// TIA Portal project "XSFW_TIA15.133301_A0" (V15.1)

(* hardware
DEVICE "S7-1200 station_1"  S7-1200 Station
   slot 0: "Rack_0"  S7-1200 Rack  Rack  V1.0
   slot 1: "PLC_1"  CPU 1214C DC/DC/DC  6ES7 214-1AG40-0XB0  V4.3
   slot 2: "DI 16x24VDC_1"  6ES7 221-1BH32-0XB0  V2.0
   slot 3: "DI 16x24VDC_2"  6ES7 221-1BH32-0XB0  V2.0
   slot 4: "DQ 16x24VDC_1"  SM 1222 DQ16 x 24VDC  6ES7 222-1BH32-0XB0  V2.0
*)

// ===== PLC "PLC_1"  CPU 1214C DC/DC/DC =====

VAR_GLOBAL   // PLC tag table "Tabla de variables_1"
   "iPul_ParEmergencia" AT %I0.0 : Bool;
   "iSel_CicloManual" AT %I0.1 : Bool;
   "iSel_CicloAuto" AT %I0.2 : Bool;
   "iSel_AvanzCamaRolos1" AT %I0.3 : Bool;
   "iSel_RetroCamaRolos1" AT %I0.4 : Bool;
   "iSel_AvanzCamaRolos2" AT %I0.5 : Bool;
   "iSel_RetroCamaRolos2" AT %I0.6 : Bool;
   "iReserva1" AT %I0.7 : Bool;
   "iProt_TermicaRolos" AT %I1.0 : Bool;
   "iStart_CicloDesdeSoldad" AT %I1.1 : Bool;
   "iSns_PresAire" AT %I1.2 : Bool;
   "iReserva2" AT %I1.3 : Bool;
   "iReserva3" AT %I1.4 : Bool;
   "iReserva4" AT %I1.5 : Bool;
   "iSns_ElevArriba" AT %I2.0 : Bool;
   "iSns_ElevAbajo" AT %I2.1 : Bool;
   "iSns_ElevNormal" AT %I2.2 : Bool;
   "iSns_ElevRotado" AT %I2.3 : Bool;
   "iSns_PreseProduc" AT %I2.4 : Bool;
   "iSns_CR1LadoTableroArri" AT %I2.5 : Bool;
   "iSns_CR1LadoTableroAbaj" AT %I2.6 : Bool;
   "iSns_RegAlturaPaq" AT %I2.7 : Bool;
   "iSns_CR1LadoOpuesArri" AT %I3.0 : Bool;
   "iSns_CR1LadoOpuesAbaj" AT %I3.1 : Bool;
   "iSns_PreseProducSalida1" AT %I3.2 : Bool;
   "iSns_PreseProducSalida2" AT %I3.3 : Bool;
   "iPul_StartCiclo" AT %I3.4 : Bool;
   "iSel_HabRuedExtrac" AT %I3.5 : Bool;
   "iPul_MarchRuedExtrac" AT %I3.6 : Bool;
   "iReserva5" AT %I3.7 : Bool;
   "iSel_HabRuedIntroduc" AT %I4.0 : Bool;
   "iPul_MarchRuedIntroduc" AT %I4.1 : Bool;
END_VAR

ORGANIZATION_BLOCK "Main"   // OB1, LAD, ProgramCycle
TITLE = "Main Program Sweep (Cycle)"
{ S7_Optimized_Access := 'TRUE' }
VERSION : 0.1
   VAR_INPUT
      Initial_Call : Bool;   // Initial call of this OB
      Remanence : Bool;   // =True, if remanent data are available
   END_VAR
BEGIN
END_ORGANIZATION_BLOCK